// Mitsubishi GX Works2 project: v04   PLC: Q02/Q02H

PROGRAM MAIN
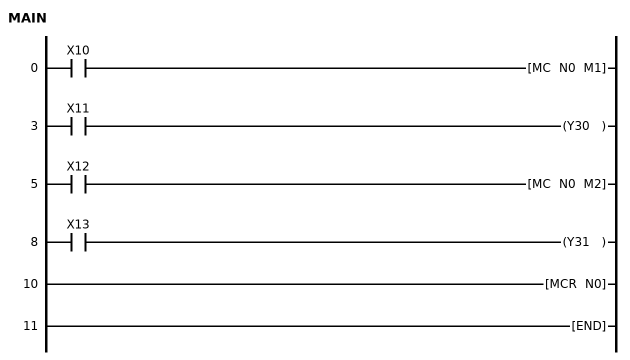
0     LD      X10
      MC      N0 M1
3     LD      X11
      OUT     Y30
5     LD      X12
      MC      N0 M2
8     LD      X13
      OUT     Y31
10    MCR     N0
11    END
END_PROGRAM
